// Mitsubishi GX Works2 project: 機電整合丙級第五題-ST   PLC: FX3U/FX3UC

// task Task_01 (event TRUE, interval 0, priority 31): POU_01

PROGRAM POU_01
VAR
  wProgramStep : INT;
  bM17 : BOOL;
  bM24 : BOOL;
  bM44 : BOOL;
  bM123 : BOOL;
  tdT22 : TON;
  tdT123 : TON;
  wMaterialType : INT;
  tdT0 : TON;
  tdT26 : TON;
  tdT211 : TON;
  bM14 : BOOL;
  bM15 : BOOL;
  tdT1 : TON;
  tdT100 : TON;
  tdT101 : TON;
END_VAR
(* 機電整合丙級術科第五題
   Author: Steven Luo
   Date: 2018/09/26
*)

IF M8002 OR NOT X17 THEN
	wProgramStep := 0;
	ZRST(TRUE, Y0, Y17);
	bM17 := FALSE;
	bM123 := FALSE;
END_IF;

IF NOT X17 THEN (* 按下急停 *)
	bM17 := TRUE;
END_IF;

IF X17 AND bM17 THEN (* 放開急停，等待復歸 *)
	tdT1(IN := FALSE);
	wProgramStep := 122;
END_IF;

IF M8002 THEN
	wProgramStep := 21;
END_IF;

IF bM123 THEN (* 黃燈閃爍 *)
	tdT100(IN := NOT tdT101.Q, PT := T#500ms);
	tdT101(IN := tdT100.Q, PT := T#500ms);
	Y16 := tdT100.Q;
ELSE
	RST(TRUE, Y16);
END_IF;

IF X14 THEN (* 指定功能 *)
	bM14 := TRUE;
ELSE
	IF wProgramStep = 215 THEN
		bM14 := FALSE;
	END_IF;
END_IF;

IF X15 THEN (* 連續循環 *)
	bM15 := TRUE;
ELSE
	bM15 := FALSE;
END_IF;

CASE wProgramStep OF
	21:
		IF X0 AND X2 AND X4 AND X5 THEN
			SET(TRUE, Y17); (* 待機，綠燈亮、紅燈滅 *)
			RST(TRUE, Y15);
			wMaterialType := 0;
			bM123 := FALSE;
			bM24 := FALSE;
			bM44 := FALSE;
		END_IF;
		IF X13 AND X17 AND X10 AND X16 THEN (* 工作模式、按下啟動鈕 *)
			tdT123(IN := FALSE);
			tdT0(IN := FALSE);
			tdT22(IN := FALSE);
			tdT26(IN := FALSE);
			tdT211(IN := FALSE);
			SET(TRUE, Y15); (* 紅燈亮、綠燈滅 *)
			RST(TRUE, Y17);
			wProgramStep := 22;
		END_IF;
	22:
		IF X10 THEN (* 有料 *)
			tdT22(IN := TRUE, PT := T#2s);
		END_IF;
		IF tdT22.Q THEN
			SET(TRUE, Y0); (* 頂料缸下降 *)
			tdT0(IN := TRUE, PT := T#2s);
		END_IF;
		IF tdT0.Q THEN
			IF X11 AND NOT X12 THEN
				wMaterialType := 1; (* 圓形料 *)
			ELSIF X11 AND X12 THEN
				wMaterialType := 2; (* 方塑料 *)
			ELSIF NOT X11 AND X12 THEN
				wMaterialType := 3; (* 方鋁料 *)
			END_IF;
			wProgramStep := 23;
		END_IF;
	23:
		RST(TRUE, Y0); (* 頂料缸上升 *)
		IF X0 THEN
			wProgramStep := 24;
		END_IF;
	24:
		SET(TRUE, Y1); (* 水平缸伸出 *)
		IF X1 THEN
			RST(TRUE, Y1);
			wProgramStep := 25;
		END_IF;
	25:
		SET(TRUE, Y3); (* 垂直缸下降 *)
		IF X3 THEN
			wProgramStep := 26;
		END_IF;
	26:
		SET(TRUE, Y10); (* 夾爪閉合 *)
		tdT26(IN := TRUE, PT := T#1s); (* 計時一秒 *)
		IF tdT26.Q THEN
			wProgramStep := 27;
		END_IF;
	27:
		RST(TRUE, Y3); (* 垂直缸上升 *)
		IF X4 THEN
			wProgramStep := 28;
		END_IF;
	28:
		SET(TRUE, Y2); (* 水平缸縮回 *)
		IF X2 THEN
			RST(TRUE, Y2);
			wProgramStep := 29;
		END_IF;
	29:
		SET(TRUE, Y5); (* 整列盤前進 *)
		IF X5 THEN (* 格位0 *)
			IF wMaterialType = 1 THEN (* 圓形料 *)
				wProgramStep := 210;
			END_IF;
		ELSIF X6 THEN (* 格位2 *)
			IF bM14 THEN (* 指定功能 *)
				IF wMaterialType = 2 THEN (* 方塑料 *)
					wProgramStep := 210;
				END_IF;
			ELSE
				IF wMaterialType = 3 THEN (* 方鋁料 *)
					wProgramStep := 210;
				END_IF;
			END_IF;
		ELSIF X7 THEN (* 格位3 *)
			IF bM14 THEN (* 指定功能 *)
				IF wMaterialType = 3 THEN (* 方鋁料 *)
					wProgramStep := 210;
				END_IF;
			ELSE
				IF wMaterialType = 2 THEN (* 方塑料 *)
					wProgramStep := 210;
				END_IF;
			END_IF;
		END_IF;
	122:
		IF NOT X13 AND X16 THEN (* 復歸模式、按下復歸開關 *)
			bM17 := FALSE;
			wProgramStep := 123;
		END_IF;
	123:
		SET(TRUE, Y11); (* 夾爪打開 *)
		tdT1(IN := TRUE, PT := T#1s); (* 計時一秒 *)
		IF tdT1.Q THEN
			RST(TRUE, Y11);
			bM123 := TRUE;
			tdT123(IN := TRUE, PT := T#3s); (* 計時三秒 *)
			SET(TRUE, Y2); (* 水平缸縮回 *)
			IF X2 THEN
				RST(TRUE, Y2);
			END_IF;
			IF tdT123.Q THEN
				wProgramStep := 124;
			END_IF;
		END_IF;
	124:
		SET(TRUE, Y6); (* 整列盤後退 *)
		IF X5 THEN (* 格位0 *)
			RST(TRUE, Y6);
			wProgramStep := 21;
		END_IF;
	210:
		RST(TRUE, Y5); (* 整列盤馬達停止 *)
		SET(TRUE, Y3); (* 垂直缸下降 *)
		IF X3 THEN
			wProgramStep := 211;
		END_IF;
	211:
		RST(TRUE, Y10);
		SET(TRUE, Y11); (* 夾爪打開 *)
		tdT211(IN := TRUE, PT := T#1s); (* 計時一秒 *)
		IF tdT211.Q THEN
			RST(TRUE, Y11);
			wProgramStep := 213;
		END_IF;
	213:
		RST(TRUE, Y3); (*垂直缸上升 *)
		IF X4 THEN
			wProgramStep := 214;
		END_IF;
	214:
		SET(TRUE, Y6); (* 整列盤後退 *)
		IF X5 THEN (* 格位0 *)
			RST(TRUE, Y6);
			wProgramStep := 215;
		END_IF;
	215:
		IF bM14 OR bM15 THEN (* 指定功能、連續循環 *)
			tdT0(IN := FALSE);
			tdT22(IN := FALSE);
			tdT26(IN := FALSE);
			tdT211(IN := FALSE);
			wProgramStep := 22;
		ELSE (* 單一循環 *)
			wProgramStep := 21;
		END_IF;
	ELSE
	;
END_CASE;
END_PROGRAM
